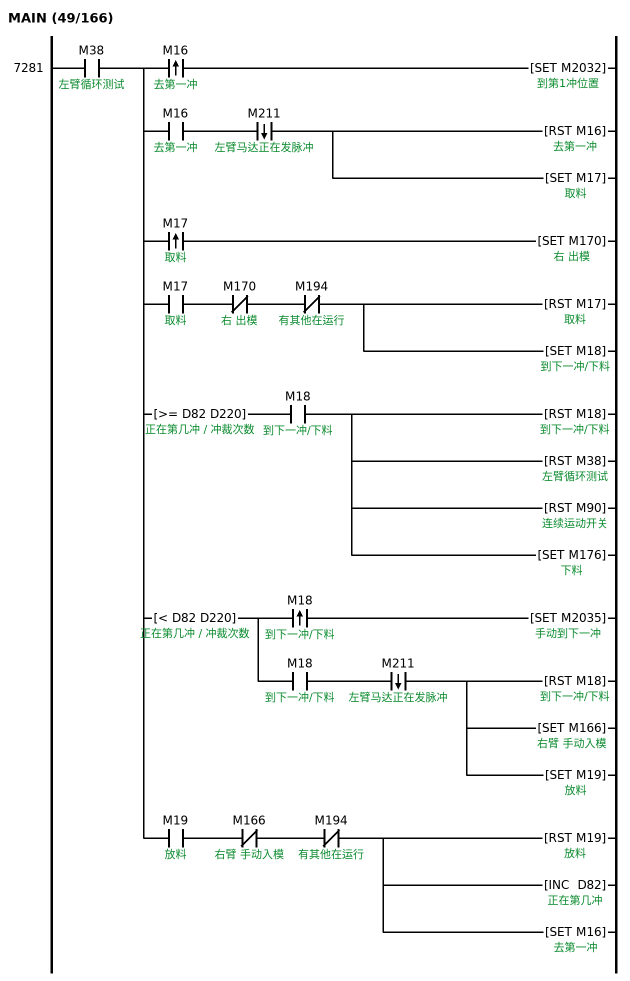
[picture p48: ladder of MAIN, rungs at steps 7281 to 7281]
7281  LD      M38  ; 左臂循环测试
      MPS
      ANDP    M16  ; 去第一冲
      SET     M2032  ; 到第1冲位置
      MRD
      AND     M16  ; 去第一冲
      ANDF    M211  ; 左臂马达正在发脉冲
      RST     M16  ; 去第一冲
      SET     M17  ; 取料
      MRD
      ANDP    M17  ; 取料
      SET     M170  ; 右 出模
      MRD
      AND     M17  ; 取料
      ANI     M170  ; 右 出模
      ANI     M194  ; 有其他在运行
      RST     M17  ; 取料
      SET     M18  ; 到下一冲/下料
      MRD
      AND>=   D82 D220  ; 正在第几冲 / 冲裁次数
      AND     M18  ; 到下一冲/下料
      RST     M18  ; 到下一冲/下料
      RST     M38  ; 左臂循环测试
      RST     M90  ; 连续运动开关
      SET     M176  ; 下料
      MRD
      AND<    D82 D220  ; 正在第几冲 / 冲裁次数
      MPS
      ANDP    M18  ; 到下一冲/下料
      SET     M2035  ; 手动到下一冲
      MPP
      AND     M18  ; 到下一冲/下料
      ANDF    M211  ; 左臂马达正在发脉冲
      RST     M18  ; 到下一冲/下料
      SET     M166  ; 右臂 手动入模
      SET     M19  ; 放料
      MPP
      AND     M19  ; 放料
      ANI     M166  ; 右臂 手动入模
      ANI     M194  ; 有其他在运行
      RST     M19  ; 放料
      INC     D82
      SET     M16  ; 去第一冲
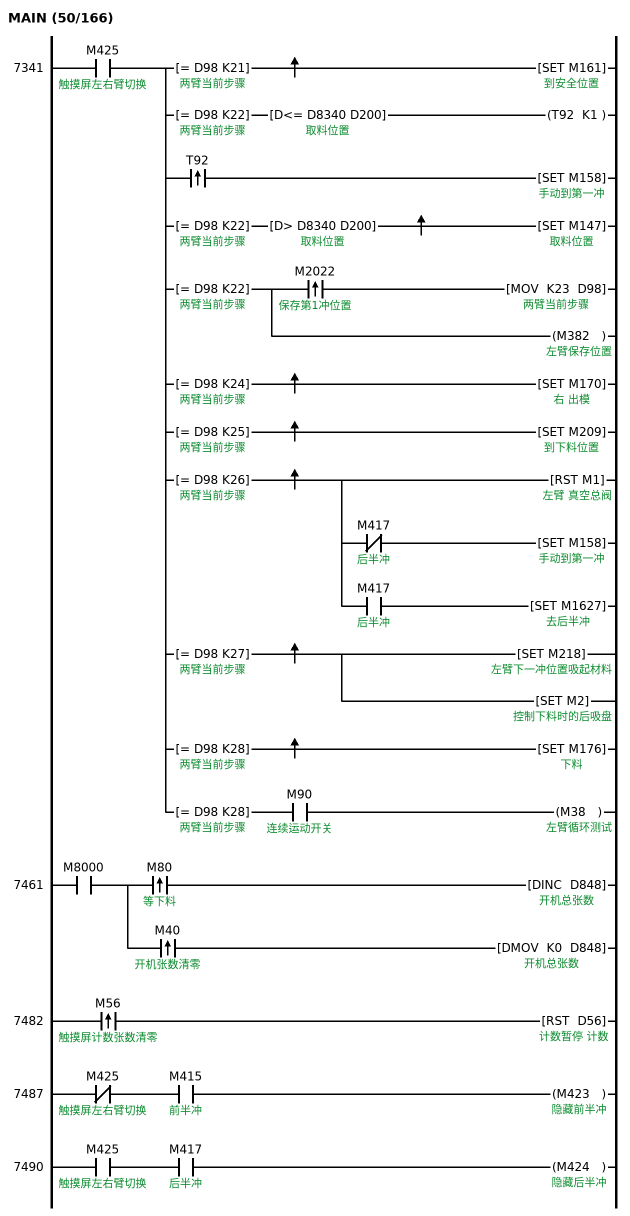
7341  LD      M425  ; 触摸屏左右臂切换
      MPS
      AND=    D98 K21  ; 两臂当前步骤
      MEP
      SET     M161  ; 到安全位置
      MRD
      AND=    D98 K22  ; 两臂当前步骤
      ANDD<=  D8340 D200  ; 取料位置
      OUT     T92 K1
      MRD
      ANDP    T92
      SET     M158  ; 手动到第一冲
      MRD
      AND=    D98 K22  ; 两臂当前步骤
      ANDD>   D8340 D200  ; 取料位置
      MEP
      SET     M147  ; 取料位置
      MRD
      AND=    D98 K22  ; 两臂当前步骤
      MPS
      ANDP    M2022  ; 保存第1冲位置
      MOV     K23 D98
      MPP
      OUT     M382  ; 左臂保存位置
      MRD
      AND=    D98 K24  ; 两臂当前步骤
      MEP
      SET     M170  ; 右 出模
      MRD
      AND=    D98 K25  ; 两臂当前步骤
      MEP
      SET     M209  ; 到下料位置
      MRD
      AND=    D98 K26  ; 两臂当前步骤
      MEP
      RST     M1  ; 左臂 真空总阀
      MPS
      ANI     M417  ; 后半冲
      SET     M158  ; 手动到第一冲
      MPP
      AND     M417  ; 后半冲
      SET     M1627  ; 去后半冲
      MRD
      AND=    D98 K27  ; 两臂当前步骤
      MEP
      SET     M218  ; 左臂下一冲位置吸起材料
      SET     M2  ; 控制下料时的后吸盘
      MRD
      AND=    D98 K28  ; 两臂当前步骤
      MEP
      SET     M176  ; 下料
      MPP
      AND=    D98 K28  ; 两臂当前步骤
      AND     M90  ; 连续运动开关
      OUT     M38  ; 左臂循环测试
7461  LD      M8000
      MPS
      ANDP    M80  ; 等下料
      DINC    D848
      MPP
      ANDP    M40  ; 开机张数清零
      DMOV    K0 D848
7482  LDP     M56  ; 触摸屏计数张数清零
      RST     D56  ; 计数暂停 计数
7487  LDI     M425  ; 触摸屏左右臂切换
      AND     M415  ; 前半冲
      OUT     M423  ; 隐藏前半冲
7490  LD      M425  ; 触摸屏左右臂切换
      AND     M417  ; 后半冲
      OUT     M424  ; 隐藏后半冲
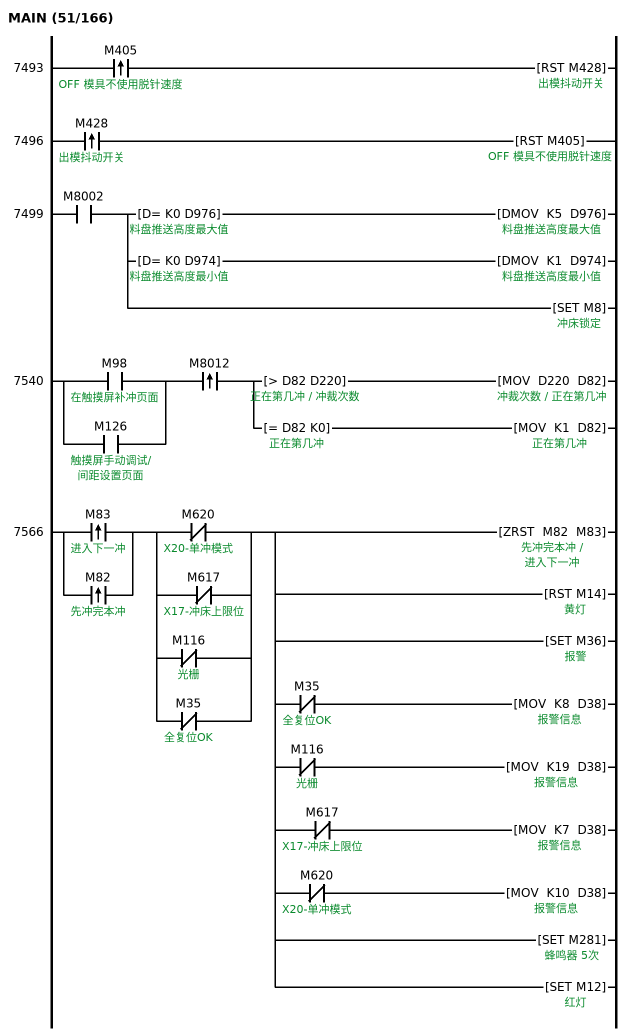
7493  LDP     M405  ; OFF 模具不使用脱针速度
      RST     M428  ; 出模抖动开关
7496  LDP     M428  ; 出模抖动开关
      RST     M405  ; OFF 模具不使用脱针速度
7499  LD      M8002
      MPS
      ANDD=   K0 D976  ; 料盘推送高度最大值
      DMOV    K5 D976
      MRD
      ANDD=   K0 D974  ; 料盘推送高度最小值
      DMOV    K1 D974
      MPP
      SET     M8  ; 冲床锁定
7540  LD      M98  ; 在触摸屏补冲页面
      OR      M126  ; 触摸屏手动调试/间距设置页面
      ANDP    M8012
      MPS
      AND>    D82 D220  ; 正在第几冲 / 冲裁次数
      MOV     D220 D82
      MPP
      AND=    D82 K0  ; 正在第几冲
      MOV     K1 D82
7566  LDP     M83  ; 进入下一冲
      ORP     M82  ; 先冲完本冲
      LDI     M620  ; X20-单冲模式
      ORI     M617  ; X17-冲床上限位
      ORI     M116  ; 光栅
      ORI     M35  ; 全复位OK
      ANB
      ZRST    M82 M83
      RST     M14  ; 黄灯
      SET     M36  ; 报警
      MPS
      ANI     M35  ; 全复位OK
      MOV     K8 D38
      MRD
      ANI     M116  ; 光栅
      MOV     K19 D38
      MRD
      ANI     M617  ; X17-冲床上限位
      MOV     K7 D38
      MRD
      ANI     M620  ; X20-单冲模式
      MOV     K10 D38
      MPP
      SET     M281  ; 蜂鸣器 5次
      SET     M12  ; 红灯
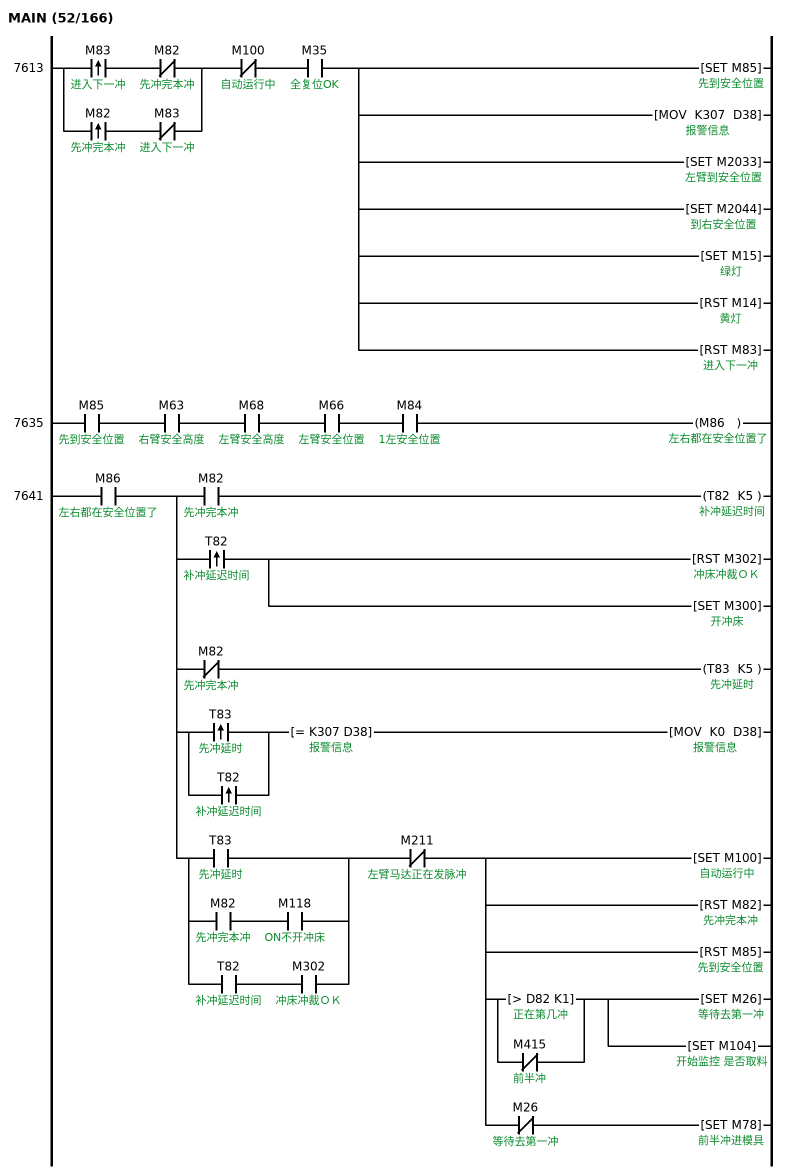
7613  LDP     M83  ; 进入下一冲
      ANI     M82  ; 先冲完本冲
      LDP     M82  ; 先冲完本冲
      ANI     M83  ; 进入下一冲
      ORB
      ANI     M100  ; 自动运行中
      AND     M35  ; 全复位OK
      SET     M85  ; 先到安全位置
      MOV     K307 D38
      SET     M2033  ; 左臂到安全位置
      SET     M2044  ; 到右安全位置
      SET     M15  ; 绿灯
      RST     M14  ; 黄灯
      RST     M83  ; 进入下一冲
7635  LD      M85  ; 先到安全位置
      AND     M63  ; 右臂安全高度
      AND     M68  ; 左臂安全高度
      AND     M66  ; 左臂安全位置
      AND     M84  ; 1左安全位置
      OUT     M86  ; 左右都在安全位置了
7641  LD      M86  ; 左右都在安全位置了
      MPS
      AND     M82  ; 先冲完本冲
      OUT     T82 K5  ; 补冲延迟时间
      MRD
      ANDP    T82  ; 补冲延迟时间
      RST     M302  ; 冲床冲裁ＯＫ
      SET     M300  ; 开冲床
      MRD
      ANI     M82  ; 先冲完本冲
      OUT     T83 K5  ; 先冲延时
      MRD
      LDP     T83  ; 先冲延时
      ORP     T82  ; 补冲延迟时间
      ANB
      AND=    K307 D38  ; 报警信息
      MOV     K0 D38
      MPP
      LD      T83  ; 先冲延时
      LD      M82  ; 先冲完本冲
      AND     M118  ; ON不开冲床
      ORB
      LD      T82  ; 补冲延迟时间
      AND     M302  ; 冲床冲裁ＯＫ
      ORB
      ANB
      ANI     M211  ; 左臂马达正在发脉冲
      SET     M100  ; 自动运行中
      RST     M82  ; 先冲完本冲
      RST     M85  ; 先到安全位置
      MPS
      LD>     D82 K1  ; 正在第几冲
      ORI     M415  ; 前半冲
      ANB
      SET     M26  ; 等待去第一冲
      SET     M104  ; 开始监控 是否取料
      MPP
      ANI     M26  ; 等待去第一冲
      SET     M78  ; 前半冲进模具
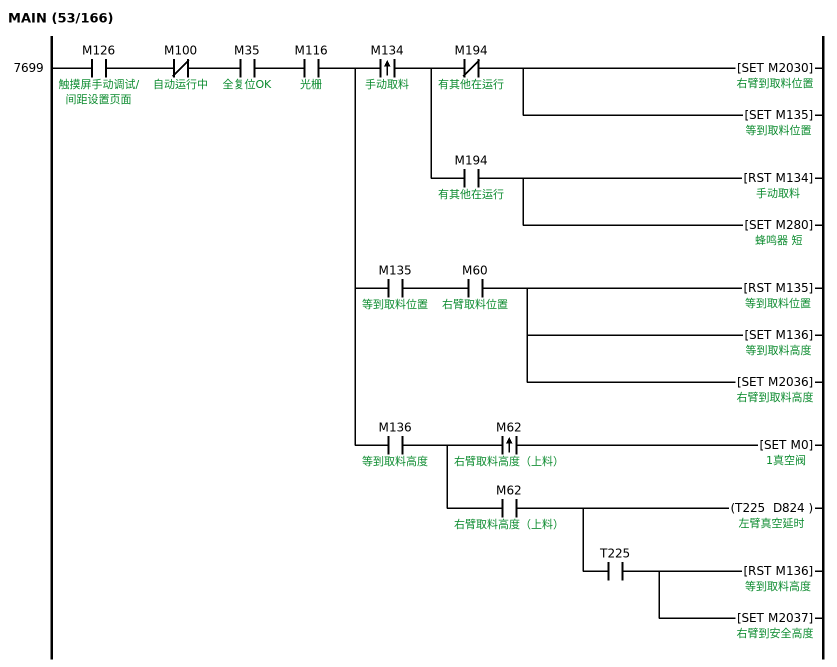
7699  LD      M126  ; 触摸屏手动调试/间距设置页面
      ANI     M100  ; 自动运行中
      AND     M35  ; 全复位OK
      AND     M116  ; 光栅
      MPS
      ANDP    M134  ; 手动取料
      MPS
      ANI     M194  ; 有其他在运行
      SET     M2030  ; 右臂到取料位置
      SET     M135  ; 等到取料位置
      MPP
      AND     M194  ; 有其他在运行
      RST     M134  ; 手动取料
      SET     M280  ; 蜂鸣器 短
      MRD
      AND     M135  ; 等到取料位置
      AND     M60  ; 右臂取料位置
      RST     M135  ; 等到取料位置
      SET     M136  ; 等到取料高度
      SET     M2036  ; 右臂到取料高度
      MPP
      AND     M136  ; 等到取料高度
      MPS
      ANDP    M62  ; 右臂取料高度（上料）
      SET     M0  ; 1真空阀
      MPP
      AND     M62  ; 右臂取料高度（上料）
      OUT     T225 D824  ; 左臂真空延时
      AND     T225
      RST     M136  ; 等到取料高度
      SET     M2037  ; 右臂到安全高度
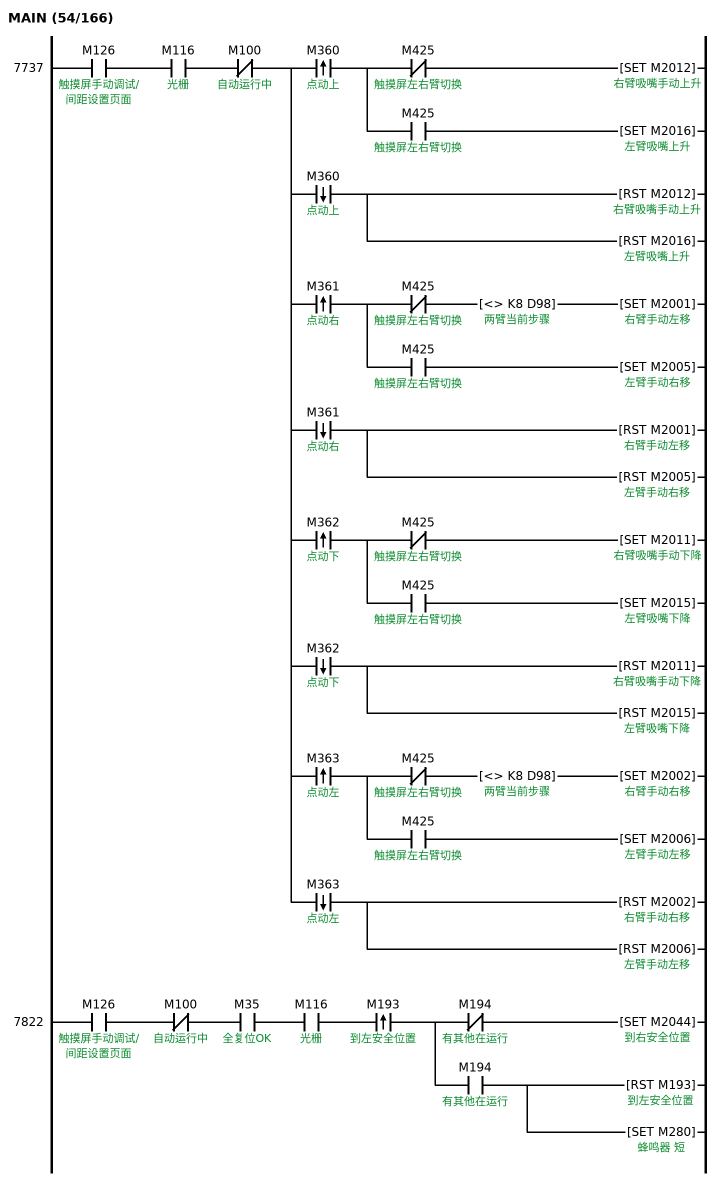
7737  LD      M126  ; 触摸屏手动调试/间距设置页面
      AND     M116  ; 光栅
      ANI     M100  ; 自动运行中
      MPS
      ANDP    M360  ; 点动上
      MPS
      ANI     M425  ; 触摸屏左右臂切换
      SET     M2012  ; 右臂吸嘴手动上升
      MPP
      AND     M425  ; 触摸屏左右臂切换
      SET     M2016  ; 左臂吸嘴上升
      MRD
      ANDF    M360  ; 点动上
      RST     M2012  ; 右臂吸嘴手动上升
      RST     M2016  ; 左臂吸嘴上升
      MRD
      ANDP    M361  ; 点动右
      MPS
      ANI     M425  ; 触摸屏左右臂切换
      AND<>   K8 D98  ; 两臂当前步骤
      SET     M2001  ; 右臂手动左移
      MPP
      AND     M425  ; 触摸屏左右臂切换
      SET     M2005  ; 左臂手动右移
      MRD
      ANDF    M361  ; 点动右
      RST     M2001  ; 右臂手动左移
      RST     M2005  ; 左臂手动右移
      MRD
      ANDP    M362  ; 点动下
      MPS
      ANI     M425  ; 触摸屏左右臂切换
      SET     M2011  ; 右臂吸嘴手动下降
      MPP
      AND     M425  ; 触摸屏左右臂切换
      SET     M2015  ; 左臂吸嘴下降
      MRD
      ANDF    M362  ; 点动下
      RST     M2011  ; 右臂吸嘴手动下降
      RST     M2015  ; 左臂吸嘴下降
      MRD
      ANDP    M363  ; 点动左
      MPS
      ANI     M425  ; 触摸屏左右臂切换
      AND<>   K8 D98  ; 两臂当前步骤
      SET     M2002  ; 右臂手动右移
      MPP
      AND     M425  ; 触摸屏左右臂切换
      SET     M2006  ; 左臂手动左移
      MPP
      ANDF    M363  ; 点动左
      RST     M2002  ; 右臂手动右移
      RST     M2006  ; 左臂手动左移
7822  LD      M126  ; 触摸屏手动调试/间距设置页面
      ANI     M100  ; 自动运行中
      AND     M35  ; 全复位OK
      AND     M116  ; 光栅
      ANDP    M193  ; 到左安全位置
      MPS
      ANI     M194  ; 有其他在运行
      SET     M2044  ; 到右安全位置
      MPP
      AND     M194  ; 有其他在运行
      RST     M193  ; 到左安全位置
      SET     M280  ; 蜂鸣器 短
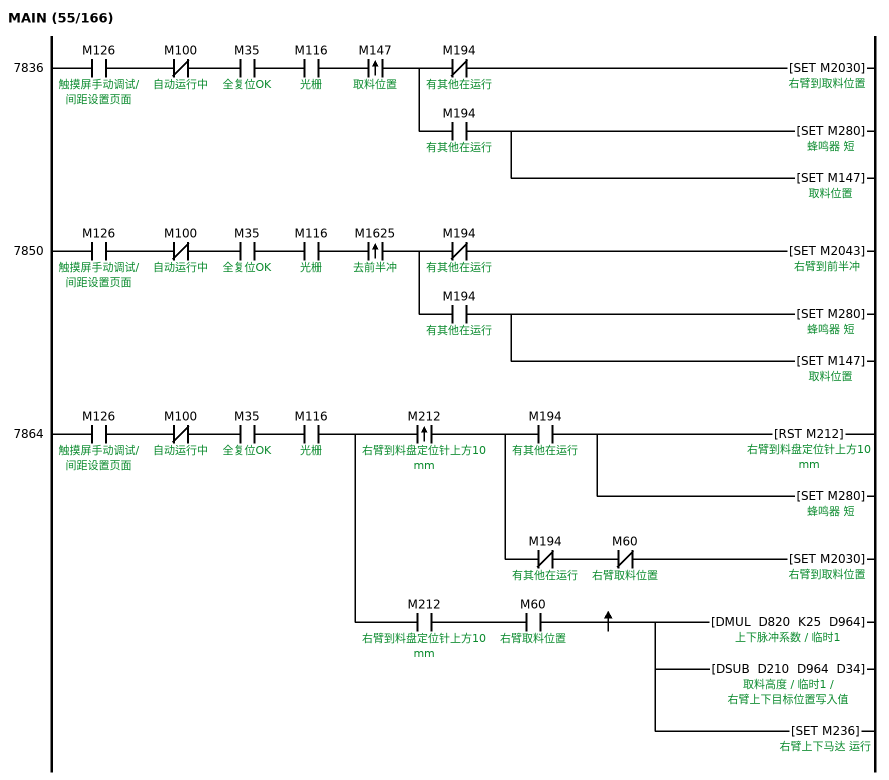
7836  LD      M126  ; 触摸屏手动调试/间距设置页面
      ANI     M100  ; 自动运行中
      AND     M35  ; 全复位OK
      AND     M116  ; 光栅
      ANDP    M147  ; 取料位置
      MPS
      ANI     M194  ; 有其他在运行
      SET     M2030  ; 右臂到取料位置
      MPP
      AND     M194  ; 有其他在运行
      SET     M280  ; 蜂鸣器 短
      SET     M147  ; 取料位置
7850  LD      M126  ; 触摸屏手动调试/间距设置页面
      ANI     M100  ; 自动运行中
      AND     M35  ; 全复位OK
      AND     M116  ; 光栅
      ANDP    M1625  ; 去前半冲
      MPS
      ANI     M194  ; 有其他在运行
      SET     M2043  ; 右臂到前半冲
      MPP
      AND     M194  ; 有其他在运行
      SET     M280  ; 蜂鸣器 短
      SET     M147  ; 取料位置
7864  LD      M126  ; 触摸屏手动调试/间距设置页面
      ANI     M100  ; 自动运行中
      AND     M35  ; 全复位OK
      AND     M116  ; 光栅
      MPS
      ANDP    M212  ; 右臂到料盘定位针上方10mm
      MPS
      AND     M194  ; 有其他在运行
      RST     M212  ; 右臂到料盘定位针上方10mm
      SET     M280  ; 蜂鸣器 短
      MPP
      ANI     M194  ; 有其他在运行
      ANI     M60  ; 右臂取料位置
      SET     M2030  ; 右臂到取料位置
      MPP
      AND     M212  ; 右臂到料盘定位针上方10mm
      AND     M60  ; 右臂取料位置
      MEP
      DMUL    D820 K25 D964
      DSUB    D210 D964 D34  ; 右臂上下目标位置写入值
      SET     M236  ; 右臂上下马达 运行
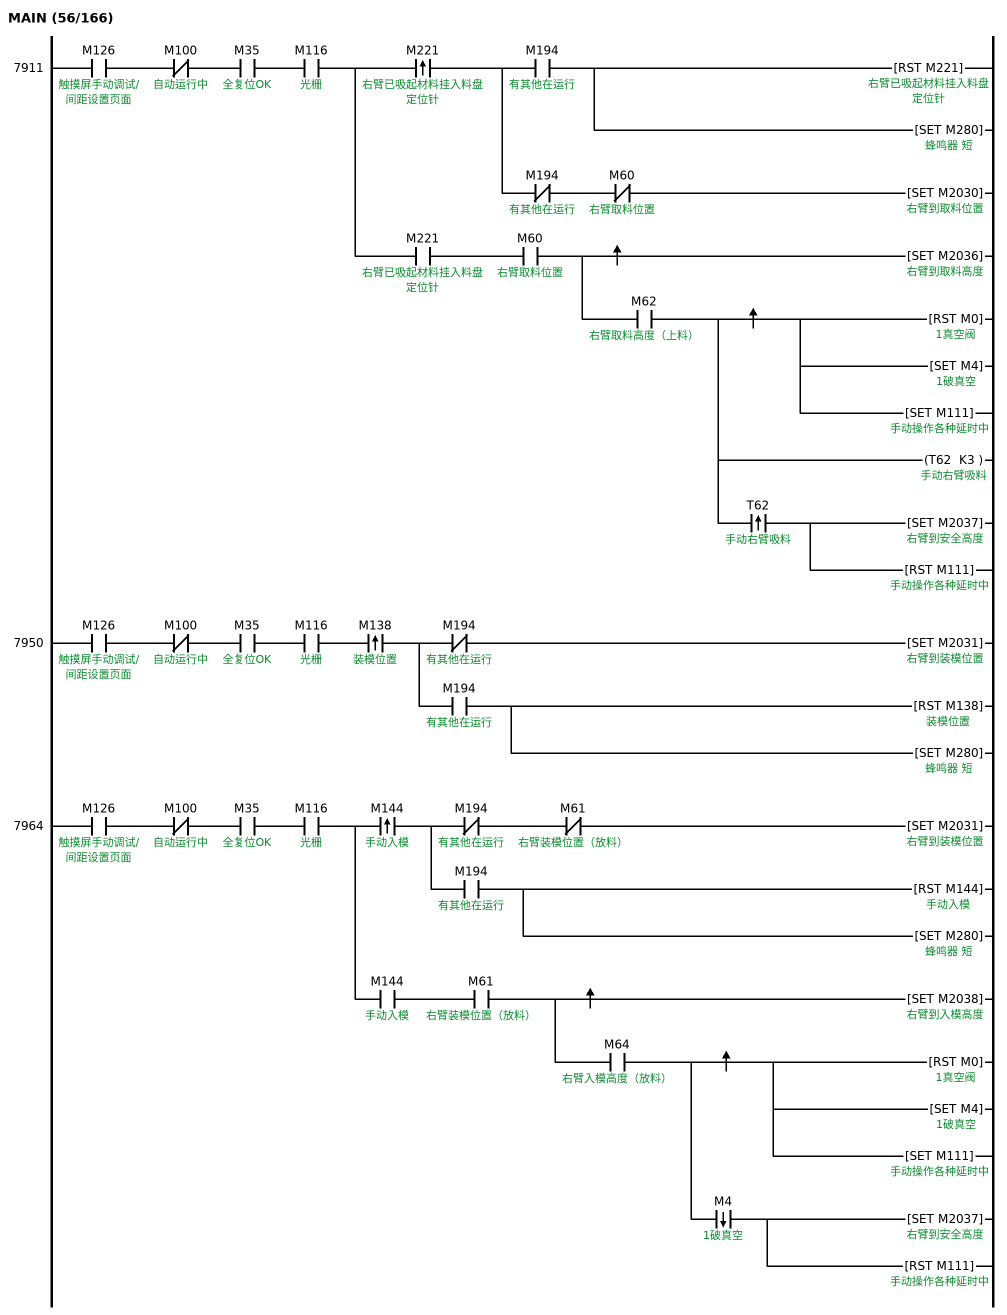
7911  LD      M126  ; 触摸屏手动调试/间距设置页面
      ANI     M100  ; 自动运行中
      AND     M35  ; 全复位OK
      AND     M116  ; 光栅
      MPS
      ANDP    M221  ; 右臂已吸起材料挂入料盘定位针
      MPS
      AND     M194  ; 有其他在运行
      RST     M221  ; 右臂已吸起材料挂入料盘定位针
      SET     M280  ; 蜂鸣器 短
      MPP
      ANI     M194  ; 有其他在运行
      ANI     M60  ; 右臂取料位置
      SET     M2030  ; 右臂到取料位置
      MPP
      AND     M221  ; 右臂已吸起材料挂入料盘定位针
      AND     M60  ; 右臂取料位置
      MPS
      MEP
      SET     M2036  ; 右臂到取料高度
      MPP
      AND     M62  ; 右臂取料高度（上料）
      MPS
      MEP
      RST     M0  ; 1真空阀
      SET     M4  ; 1破真空
      SET     M111  ; 手动操作各种延时中
      MPP
      OUT     T62 K3  ; 手动右臂吸料
      ANDP    T62  ; 手动右臂吸料
      SET     M2037  ; 右臂到安全高度
      RST     M111  ; 手动操作各种延时中
7950  LD      M126  ; 触摸屏手动调试/间距设置页面
      ANI     M100  ; 自动运行中
      AND     M35  ; 全复位OK
      AND     M116  ; 光栅
      ANDP    M138  ; 装模位置
      MPS
      ANI     M194  ; 有其他在运行
      SET     M2031  ; 右臂到装模位置
      MPP
      AND     M194  ; 有其他在运行
      RST     M138  ; 装模位置
      SET     M280  ; 蜂鸣器 短
7964  LD      M126  ; 触摸屏手动调试/间距设置页面
      ANI     M100  ; 自动运行中
      AND     M35  ; 全复位OK
      AND     M116  ; 光栅
      MPS
      ANDP    M144  ; 手动入模
      MPS
      ANI     M194  ; 有其他在运行
      ANI     M61  ; 右臂装模位置（放料）
      SET     M2031  ; 右臂到装模位置
      MPP
      AND     M194  ; 有其他在运行
      RST     M144  ; 手动入模
      SET     M280  ; 蜂鸣器 短
      MPP
      AND     M144  ; 手动入模
      AND     M61  ; 右臂装模位置（放料）
      MPS
      MEP
      SET     M2038  ; 右臂到入模高度
      MPP
      AND     M64  ; 右臂入模高度（放料）
      MPS
      MEP
      RST     M0  ; 1真空阀
      SET     M4  ; 1破真空
      SET     M111  ; 手动操作各种延时中
      MPP
      ANDF    M4  ; 1破真空
      SET     M2037  ; 右臂到安全高度
      RST     M111  ; 手动操作各种延时中
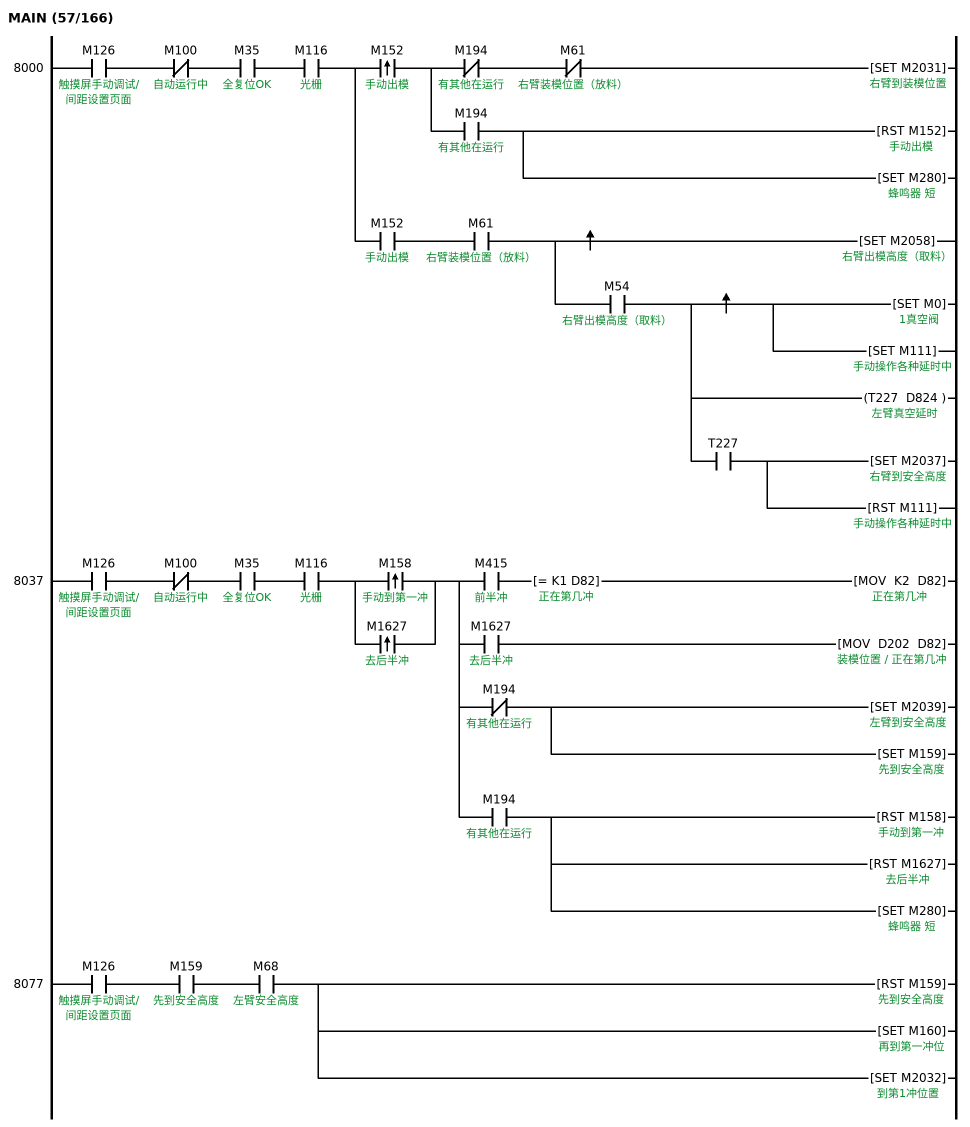
8000  LD      M126  ; 触摸屏手动调试/间距设置页面
      ANI     M100  ; 自动运行中
      AND     M35  ; 全复位OK
      AND     M116  ; 光栅
      MPS
      ANDP    M152  ; 手动出模
      MPS
      ANI     M194  ; 有其他在运行
      ANI     M61  ; 右臂装模位置（放料）
      SET     M2031  ; 右臂到装模位置
      MPP
      AND     M194  ; 有其他在运行
      RST     M152  ; 手动出模
      SET     M280  ; 蜂鸣器 短
      MPP
      AND     M152  ; 手动出模
      AND     M61  ; 右臂装模位置（放料）
      MPS
      MEP
      SET     M2058  ; 右臂出模高度（取料）
      MPP
      AND     M54  ; 右臂出模高度（取料）
      MPS
      MEP
      SET     M0  ; 1真空阀
      SET     M111  ; 手动操作各种延时中
      MPP
      OUT     T227 D824  ; 左臂真空延时
      AND     T227
      SET     M2037  ; 右臂到安全高度
      RST     M111  ; 手动操作各种延时中
8037  LD      M126  ; 触摸屏手动调试/间距设置页面
      ANI     M100  ; 自动运行中
      AND     M35  ; 全复位OK
      AND     M116  ; 光栅
      LDP     M158  ; 手动到第一冲
      ORP     M1627  ; 去后半冲
      ANB
      MPS
      AND     M415  ; 前半冲
      AND=    K1 D82  ; 正在第几冲
      MOV     K2 D82
      MRD
      AND     M1627  ; 去后半冲
      MOV     D202 D82
      MRD
      ANI     M194  ; 有其他在运行
      SET     M2039  ; 左臂到安全高度
      SET     M159  ; 先到安全高度
      MPP
      AND     M194  ; 有其他在运行
      RST     M158  ; 手动到第一冲
      RST     M1627  ; 去后半冲
      SET     M280  ; 蜂鸣器 短
8077  LD      M126  ; 触摸屏手动调试/间距设置页面
      AND     M159  ; 先到安全高度
      AND     M68  ; 左臂安全高度
      RST     M159  ; 先到安全高度
      SET     M160  ; 再到第一冲位
      SET     M2032  ; 到第1冲位置
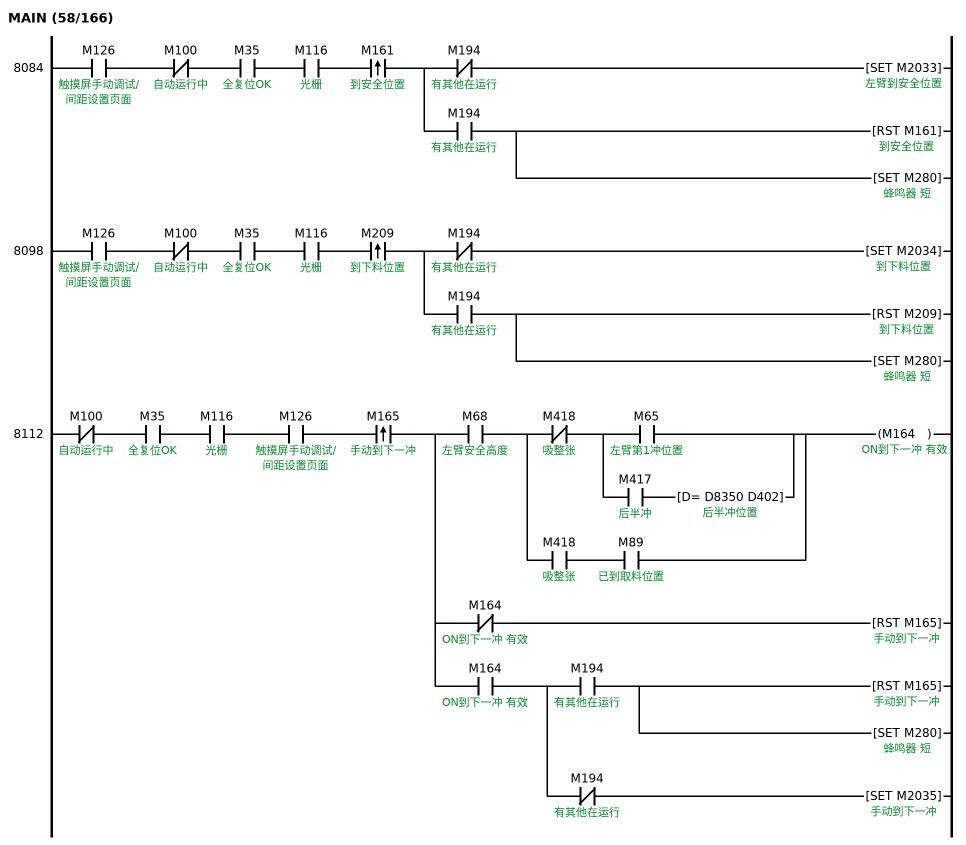
8084  LD      M126  ; 触摸屏手动调试/间距设置页面
      ANI     M100  ; 自动运行中
      AND     M35  ; 全复位OK
      AND     M116  ; 光栅
      ANDP    M161  ; 到安全位置
      MPS
      ANI     M194  ; 有其他在运行
      SET     M2033  ; 左臂到安全位置
      MPP
      AND     M194  ; 有其他在运行
      RST     M161  ; 到安全位置
      SET     M280  ; 蜂鸣器 短
8098  LD      M126  ; 触摸屏手动调试/间距设置页面
      ANI     M100  ; 自动运行中
      AND     M35  ; 全复位OK
      AND     M116  ; 光栅
      ANDP    M209  ; 到下料位置
      MPS
      ANI     M194  ; 有其他在运行
      SET     M2034  ; 到下料位置
      MPP
      AND     M194  ; 有其他在运行
      RST     M209  ; 到下料位置
      SET     M280  ; 蜂鸣器 短
8112  LDI     M100  ; 自动运行中
      AND     M35  ; 全复位OK
      AND     M116  ; 光栅
      AND     M126  ; 触摸屏手动调试/间距设置页面
      ANDP    M165  ; 手动到下一冲
      MPS
      AND     M68  ; 左臂安全高度
      LDI     M418  ; 吸整张
      LD      M65  ; 左臂第1冲位置
      LD      M417  ; 后半冲
      ANDD=   D8350 D402  ; 后半冲位置
      ORB
      ANB
      LD      M418  ; 吸整张
      AND     M89  ; 已到取料位置
      ORB
      ANB
      OUT     M164  ; ON到下一冲 有效
      MRD
      ANI     M164  ; ON到下一冲 有效
      RST     M165  ; 手动到下一冲
      MPP
      AND     M164  ; ON到下一冲 有效
      MPS
      AND     M194  ; 有其他在运行
      RST     M165  ; 手动到下一冲
      SET     M280  ; 蜂鸣器 短
      MPP
      ANI     M194  ; 有其他在运行
      SET     M2035  ; 手动到下一冲
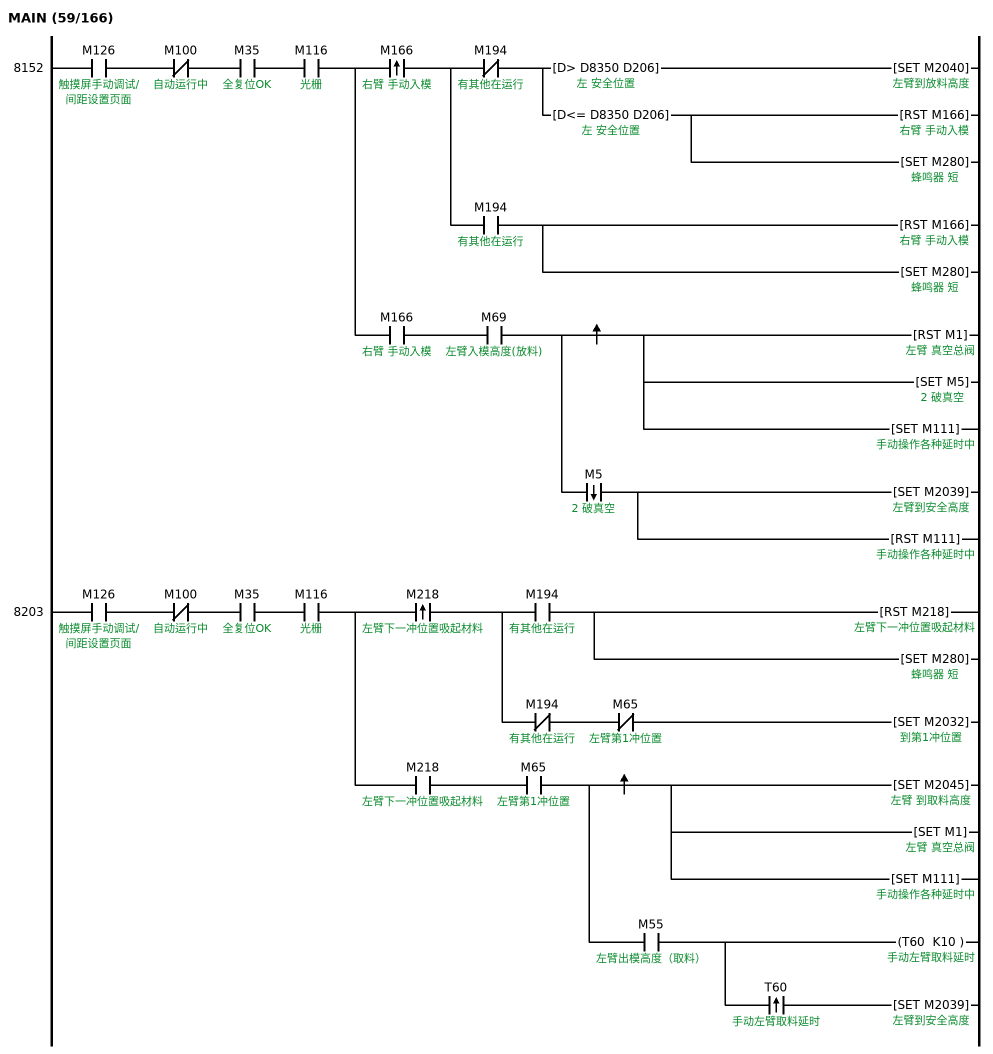
8152  LD      M126  ; 触摸屏手动调试/间距设置页面
      ANI     M100  ; 自动运行中
      AND     M35  ; 全复位OK
      AND     M116  ; 光栅
      MPS
      ANDP    M166  ; 右臂 手动入模
      MPS
      ANI     M194  ; 有其他在运行
      MPS
      ANDD>   D8350 D206  ; 左 安全位置
      SET     M2040  ; 左臂到放料高度
      MPP
      ANDD<=  D8350 D206  ; 左 安全位置
      RST     M166  ; 右臂 手动入模
      SET     M280  ; 蜂鸣器 短
      MPP
      AND     M194  ; 有其他在运行
      RST     M166  ; 右臂 手动入模
      SET     M280  ; 蜂鸣器 短
      MPP
      AND     M166  ; 右臂 手动入模
      AND     M69  ; 左臂入模高度(放料)
      MPS
      MEP
      RST     M1  ; 左臂 真空总阀
      SET     M5  ; 2 破真空
      SET     M111  ; 手动操作各种延时中
      MPP
      ANDF    M5  ; 2 破真空
      SET     M2039  ; 左臂到安全高度
      RST     M111  ; 手动操作各种延时中
8203  LD      M126  ; 触摸屏手动调试/间距设置页面
      ANI     M100  ; 自动运行中
      AND     M35  ; 全复位OK
      AND     M116  ; 光栅
      MPS
      ANDP    M218  ; 左臂下一冲位置吸起材料
      MPS
      AND     M194  ; 有其他在运行
      RST     M218  ; 左臂下一冲位置吸起材料
      SET     M280  ; 蜂鸣器 短
      MPP
      ANI     M194  ; 有其他在运行
      ANI     M65  ; 左臂第1冲位置
      SET     M2032  ; 到第1冲位置
      MPP
      AND     M218  ; 左臂下一冲位置吸起材料
      AND     M65  ; 左臂第1冲位置
      MPS
      MEP
      SET     M2045  ; 左臂 到取料高度
      SET     M1  ; 左臂 真空总阀
      SET     M111  ; 手动操作各种延时中
      MPP
      AND     M55  ; 左臂出模高度（取料）
      OUT     T60 K10  ; 手动左臂取料延时
      ANDP    T60  ; 手动左臂取料延时
      SET     M2039  ; 左臂到安全高度
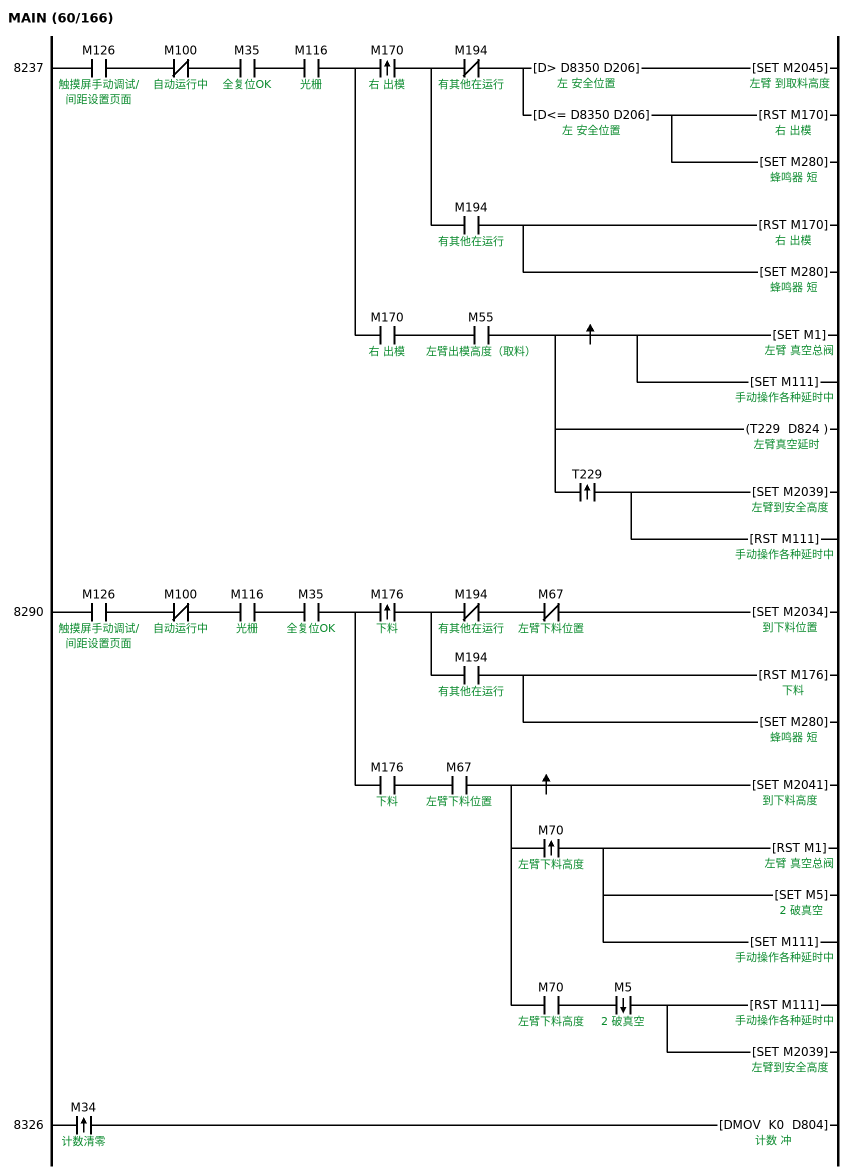
8237  LD      M126  ; 触摸屏手动调试/间距设置页面
      ANI     M100  ; 自动运行中
      AND     M35  ; 全复位OK
      AND     M116  ; 光栅
      MPS
      ANDP    M170  ; 右 出模
      MPS
      ANI     M194  ; 有其他在运行
      MPS
      ANDD>   D8350 D206  ; 左 安全位置
      SET     M2045  ; 左臂 到取料高度
      MPP
      ANDD<=  D8350 D206  ; 左 安全位置
      RST     M170  ; 右 出模
      SET     M280  ; 蜂鸣器 短
      MPP
      AND     M194  ; 有其他在运行
      RST     M170  ; 右 出模
      SET     M280  ; 蜂鸣器 短
      MPP
      AND     M170  ; 右 出模
      AND     M55  ; 左臂出模高度（取料）
      MPS
      MEP
      SET     M1  ; 左臂 真空总阀
      SET     M111  ; 手动操作各种延时中
      MPP
      OUT     T229 D824  ; 左臂真空延时
      ANDP    T229
      SET     M2039  ; 左臂到安全高度
      RST     M111  ; 手动操作各种延时中
8290  LD      M126  ; 触摸屏手动调试/间距设置页面
      ANI     M100  ; 自动运行中
      AND     M116  ; 光栅
      AND     M35  ; 全复位OK
      MPS
      ANDP    M176  ; 下料
      MPS
      ANI     M194  ; 有其他在运行
      ANI     M67  ; 左臂下料位置
      SET     M2034  ; 到下料位置
      MPP
      AND     M194  ; 有其他在运行
      RST     M176  ; 下料
      SET     M280  ; 蜂鸣器 短
      MPP
      AND     M176  ; 下料
      AND     M67  ; 左臂下料位置
      MPS
      MEP
      SET     M2041  ; 到下料高度
      MRD
      ANDP    M70  ; 左臂下料高度
      RST     M1  ; 左臂 真空总阀
      SET     M5  ; 2 破真空
      SET     M111  ; 手动操作各种延时中
      MPP
      AND     M70  ; 左臂下料高度
      ANDF    M5  ; 2 破真空
      RST     M111  ; 手动操作各种延时中
      SET     M2039  ; 左臂到安全高度
8326  LDP     M34  ; 计数清零
      DMOV    K0 D804
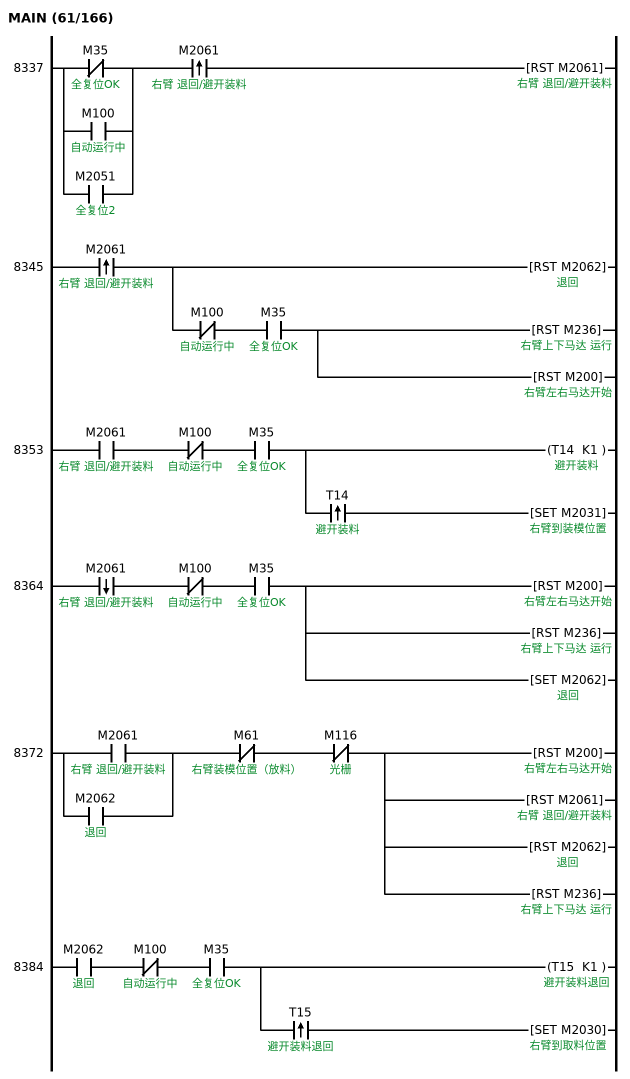
8337  LDI     M35  ; 全复位OK
      OR      M100  ; 自动运行中
      OR      M2051  ; 全复位2
      ANDP    M2061  ; 右臂 退回/避开装料
      RST     M2061  ; 右臂 退回/避开装料
8345  LDP     M2061  ; 右臂 退回/避开装料
      RST     M2062  ; 退回
      ANI     M100  ; 自动运行中
      AND     M35  ; 全复位OK
      RST     M236  ; 右臂上下马达 运行
      RST     M200  ; 右臂左右马达开始
8353  LD      M2061  ; 右臂 退回/避开装料
      ANI     M100  ; 自动运行中
      AND     M35  ; 全复位OK
      OUT     T14 K1  ; 避开装料
      ANDP    T14  ; 避开装料
      SET     M2031  ; 右臂到装模位置
8364  LDF     M2061  ; 右臂 退回/避开装料
      ANI     M100  ; 自动运行中
      AND     M35  ; 全复位OK
      RST     M200  ; 右臂左右马达开始
      RST     M236  ; 右臂上下马达 运行
      SET     M2062  ; 退回
8372  LD      M2061  ; 右臂 退回/避开装料
      OR      M2062  ; 退回
      ANI     M61  ; 右臂装模位置（放料）
      ANI     M116  ; 光栅
      RST     M200  ; 右臂左右马达开始
      RST     M2061  ; 右臂 退回/避开装料
      RST     M2062  ; 退回
      RST     M236  ; 右臂上下马达 运行
8384  LD      M2062  ; 退回
      ANI     M100  ; 自动运行中
      AND     M35  ; 全复位OK
      OUT     T15 K1  ; 避开装料退回
      ANDP    T15  ; 避开装料退回
      SET     M2030  ; 右臂到取料位置
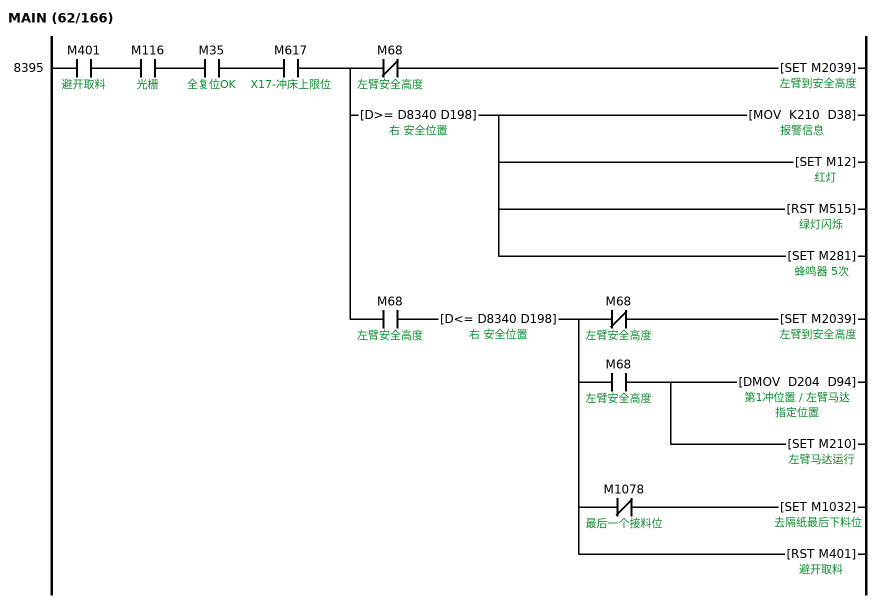
8395  LD      M401  ; 避开取料
      AND     M116  ; 光栅
      AND     M35  ; 全复位OK
      AND     M617  ; X17-冲床上限位
      MPS
      ANI     M68  ; 左臂安全高度
      SET     M2039  ; 左臂到安全高度
      MRD
      ANDD>=  D8340 D198  ; 右 安全位置
      MOV     K210 D38
      SET     M12  ; 红灯
      RST     M515  ; 绿灯闪烁
      SET     M281  ; 蜂鸣器 5次
      MPP
      AND     M68  ; 左臂安全高度
      ANDD<=  D8340 D198  ; 右 安全位置
      MPS
      ANI     M68  ; 左臂安全高度
      SET     M2039  ; 左臂到安全高度
      MRD
      AND     M68  ; 左臂安全高度
      DMOV    D204 D94
      SET     M210  ; 左臂马达运行
      MRD
      ANI     M1078  ; 最后一个接料位
      SET     M1032  ; 去隔纸最后下料位
      MPP
      RST     M401  ; 避开取料
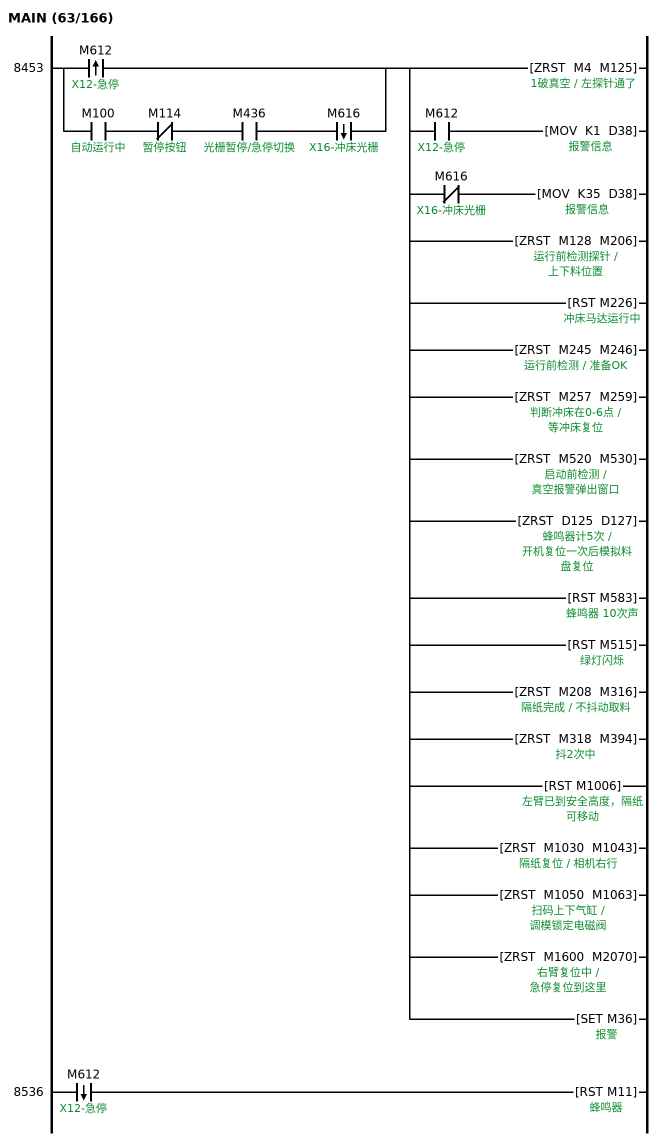
8453  LDP     M612  ; X12-急停
      LD      M100  ; 自动运行中
      ANI     M114  ; 暂停按钮
      AND     M436  ; 光栅暂停/急停切换
      ANDF    M616  ; X16-冲床光栅
      ORB
      ZRST    M4 M125
      MPS
      AND     M612  ; X12-急停
      MOV     K1 D38
      MRD
      ANI     M616  ; X16-冲床光栅
      MOV     K35 D38
      MPP
      ZRST    M128 M206  ; 上下料位置
      RST     M226  ; 冲床马达运行中
      ZRST    M245 M246  ; 运行前检测 / 准备OK
      ZRST    M257 M259  ; 判断冲床在0-6点 / 等冲床复位
      ZRST    M520 M530  ; 启动前检测
      ZRST    D125 D127  ; 蜂鸣器计5次 / 开机复位一次后模拟料盘复位
      RST     M583  ; 蜂鸣器 10次声
      RST     M515  ; 绿灯闪烁
      ZRST    M208 M316  ; 隔纸完成
      ZRST    M318 M394
      RST     M1006  ; 左臂已到安全高度，隔纸可移动
      ZRST    M1030 M1043
      ZRST    M1050 M1063
      ZRST    M1600 M2070  ; 急停复位到这里
      SET     M36  ; 报警
8536  LDF     M612  ; X12-急停
      RST     M11  ; 蜂鸣器
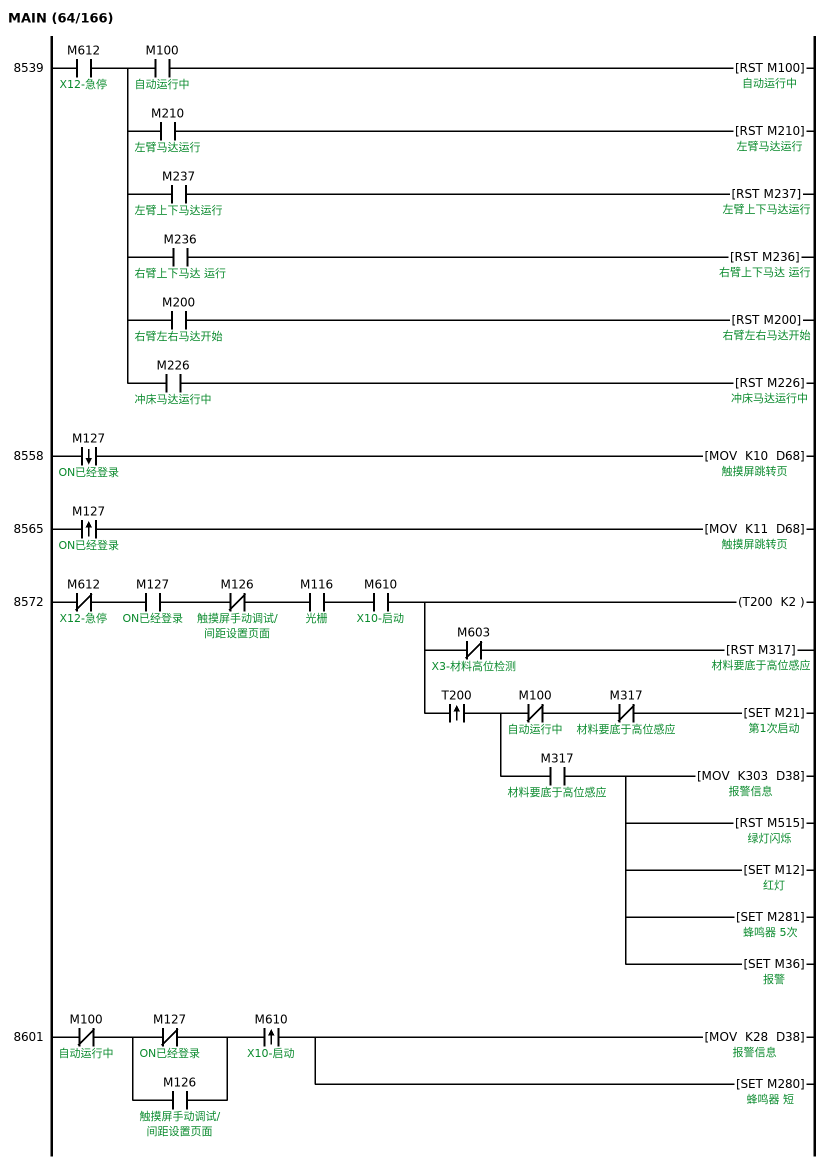
8539  LD      M612  ; X12-急停
      MPS
      AND     M100  ; 自动运行中
      RST     M100  ; 自动运行中
      MRD
      AND     M210  ; 左臂马达运行
      RST     M210  ; 左臂马达运行
      MRD
      AND     M237  ; 左臂上下马达运行
      RST     M237  ; 左臂上下马达运行
      MRD
      AND     M236  ; 右臂上下马达 运行
      RST     M236  ; 右臂上下马达 运行
      MRD
      AND     M200  ; 右臂左右马达开始
      RST     M200  ; 右臂左右马达开始
      MPP
      AND     M226  ; 冲床马达运行中
      RST     M226  ; 冲床马达运行中
8558  LDF     M127  ; ON已经登录
      MOV     K10 D68  ; 触摸屏跳转页
8565  LDP     M127  ; ON已经登录
      MOV     K11 D68
8572  LDI     M612  ; X12-急停
      AND     M127  ; ON已经登录
      ANI     M126  ; 触摸屏手动调试/间距设置页面
      AND     M116  ; 光栅
      AND     M610  ; X10-启动
      OUT     T200 K2
      MPS
      ANI     M603  ; X3-材料高位检测
      RST     M317  ; 材料要底于高位感应
      MPP
      ANDP    T200
      MPS
      ANI     M100  ; 自动运行中
      ANI     M317  ; 材料要底于高位感应
      SET     M21  ; 第1次启动
      MPP
      AND     M317  ; 材料要底于高位感应
      MOV     K303 D38
      RST     M515  ; 绿灯闪烁
      SET     M12  ; 红灯
      SET     M281  ; 蜂鸣器 5次
      SET     M36  ; 报警
8601  LDI     M100  ; 自动运行中
      LDI     M127  ; ON已经登录
      OR      M126  ; 触摸屏手动调试/间距设置页面
      ANB
      ANDP    M610  ; X10-启动
      MOV     K28 D38
      SET     M280  ; 蜂鸣器 短
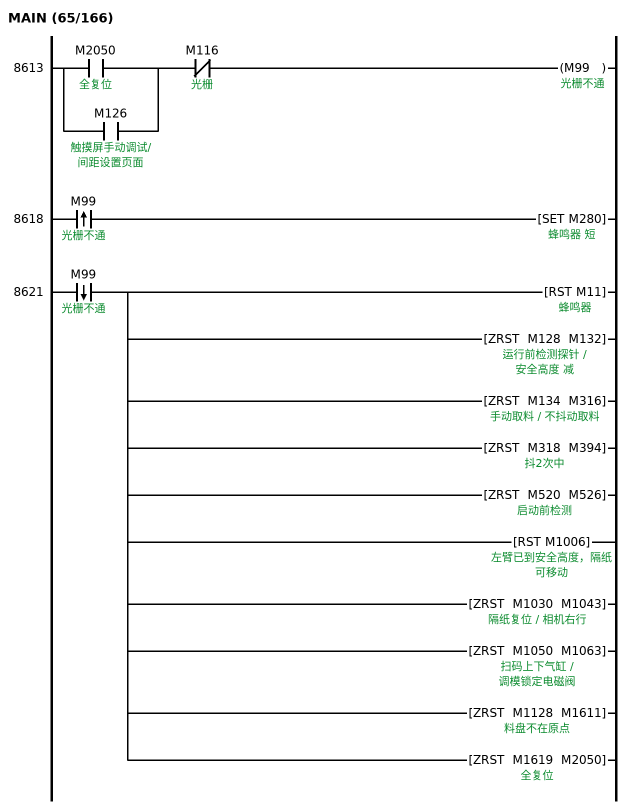
8613  LD      M2050  ; 全复位
      OR      M126  ; 触摸屏手动调试/间距设置页面
      ANI     M116  ; 光栅
      OUT     M99  ; 光栅不通
8618  LDP     M99  ; 光栅不通
      SET     M280  ; 蜂鸣器 短
8621  LDF     M99  ; 光栅不通
      RST     M11  ; 蜂鸣器
      ZRST    M128 M132
      ZRST    M134 M316
      ZRST    M318 M394
      ZRST    M520 M526
      RST     M1006  ; 左臂已到安全高度，隔纸可移动
      ZRST    M1030 M1043
      ZRST    M1050 M1063
      ZRST    M1128 M1611  ; 料盘不在原点
      ZRST    M1619 M2050
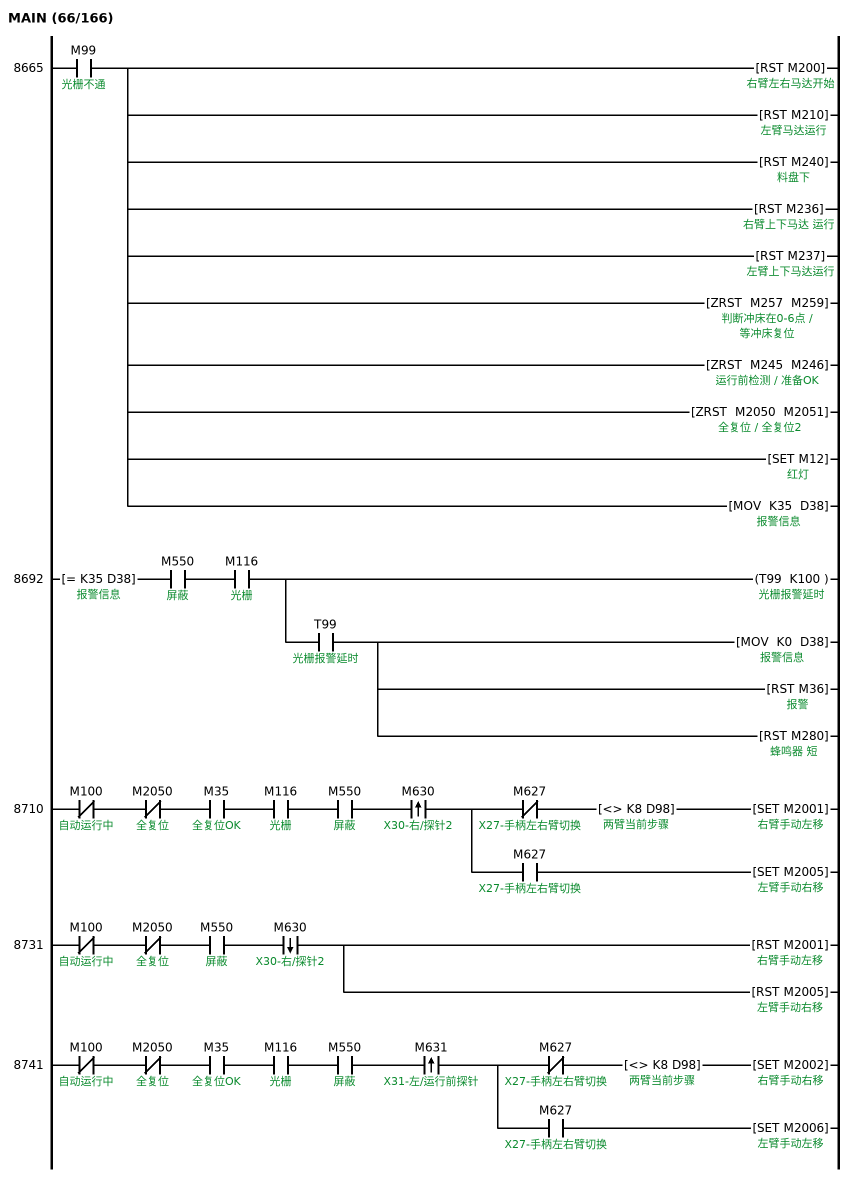
8665  LD      M99  ; 光栅不通
      RST     M200  ; 右臂左右马达开始
      RST     M210  ; 左臂马达运行
      RST     M240  ; 料盘下
      RST     M236  ; 右臂上下马达 运行
      RST     M237  ; 左臂上下马达运行
      ZRST    M257 M259
      ZRST    M245 M246
      ZRST    M2050 M2051
      SET     M12  ; 红灯
      MOV     K35 D38
8692  LD=     K35 D38  ; 报警信息
      AND     M550  ; 屏蔽
      AND     M116  ; 光栅
      OUT     T99 K100  ; 光栅报警延时
      AND     T99  ; 光栅报警延时
      MOV     K0 D38
      RST     M36  ; 报警
      RST     M280  ; 蜂鸣器 短
8710  LDI     M100  ; 自动运行中
      ANI     M2050  ; 全复位
      AND     M35  ; 全复位OK
      AND     M116  ; 光栅
      AND     M550  ; 屏蔽
      ANDP    M630  ; X30-右/探针2
      MPS
      ANI     M627  ; X27-手柄左右臂切换
      AND<>   K8 D98  ; 两臂当前步骤
      SET     M2001  ; 右臂手动左移
      MPP
      AND     M627  ; X27-手柄左右臂切换
      SET     M2005  ; 左臂手动右移
8731  LDI     M100  ; 自动运行中
      ANI     M2050  ; 全复位
      AND     M550  ; 屏蔽
      ANDF    M630  ; X30-右/探针2
      RST     M2001  ; 右臂手动左移
      RST     M2005  ; 左臂手动右移
8741  LDI     M100  ; 自动运行中
      ANI     M2050  ; 全复位
      AND     M35  ; 全复位OK
      AND     M116  ; 光栅
      AND     M550  ; 屏蔽
      ANDP    M631  ; X31-左/运行前探针
      MPS
      ANI     M627  ; X27-手柄左右臂切换
      AND<>   K8 D98  ; 两臂当前步骤
      SET     M2002  ; 右臂手动右移
      MPP
      AND     M627  ; X27-手柄左右臂切换
      SET     M2006  ; 左臂手动左移
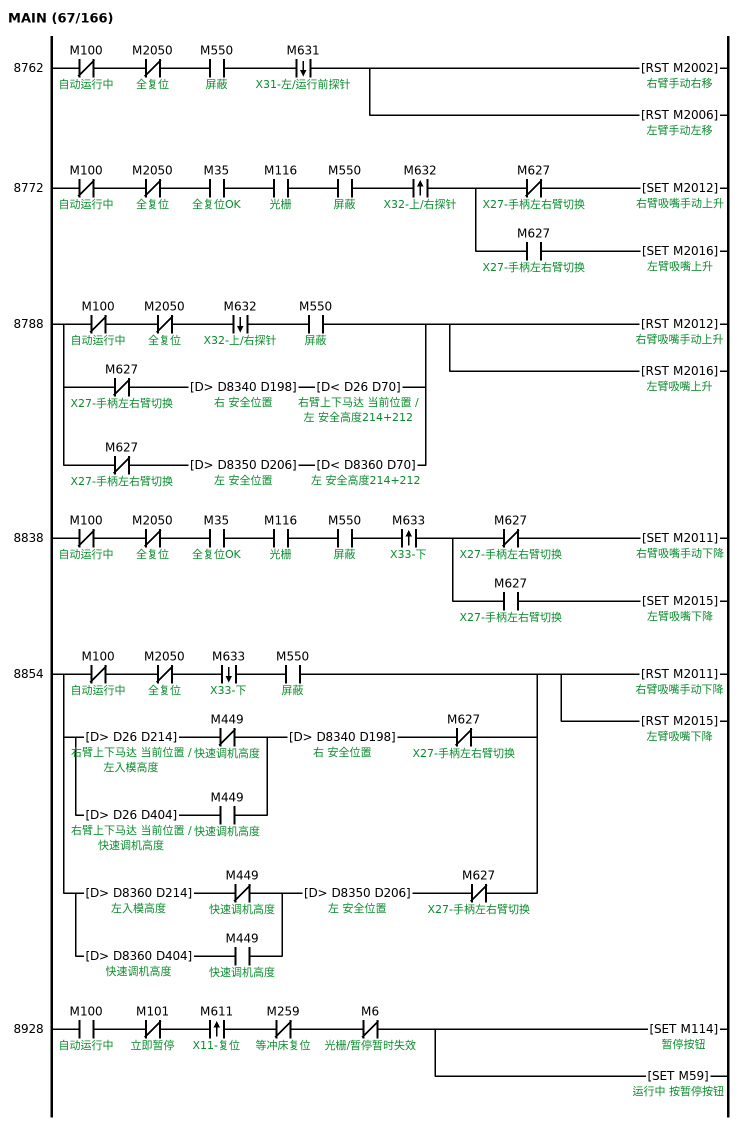
8762  LDI     M100  ; 自动运行中
      ANI     M2050  ; 全复位
      AND     M550  ; 屏蔽
      ANDF    M631  ; X31-左/运行前探针
      RST     M2002  ; 右臂手动右移
      RST     M2006  ; 左臂手动左移
8772  LDI     M100  ; 自动运行中
      ANI     M2050  ; 全复位
      AND     M35  ; 全复位OK
      AND     M116  ; 光栅
      AND     M550  ; 屏蔽
      ANDP    M632  ; X32-上/右探针
      MPS
      ANI     M627  ; X27-手柄左右臂切换
      SET     M2012  ; 右臂吸嘴手动上升
      MPP
      AND     M627  ; X27-手柄左右臂切换
      SET     M2016  ; 左臂吸嘴上升
8788  LDI     M100  ; 自动运行中
      ANI     M2050  ; 全复位
      ANDF    M632  ; X32-上/右探针
      AND     M550  ; 屏蔽
      LDI     M627  ; X27-手柄左右臂切换
      ANDD>   D8340 D198  ; 右 安全位置
      ANDD<   D26 D70  ; 右臂上下马达 当前位置 / 左 安全高度214+212
      ORB
      LDI     M627  ; X27-手柄左右臂切换
      ANDD>   D8350 D206  ; 左 安全位置
      ANDD<   D8360 D70  ; 左 安全高度214+212
      ORB
      RST     M2012  ; 右臂吸嘴手动上升
      RST     M2016  ; 左臂吸嘴上升
8838  LDI     M100  ; 自动运行中
      ANI     M2050  ; 全复位
      AND     M35  ; 全复位OK
      AND     M116  ; 光栅
      AND     M550  ; 屏蔽
      ANDP    M633  ; X33-下
      MPS
      ANI     M627  ; X27-手柄左右臂切换
      SET     M2011  ; 右臂吸嘴手动下降
      MPP
      AND     M627  ; X27-手柄左右臂切换
      SET     M2015  ; 左臂吸嘴下降
8854  LDI     M100  ; 自动运行中
      ANI     M2050  ; 全复位
      ANDF    M633  ; X33-下
      AND     M550  ; 屏蔽
      LDD>    D26 D214  ; 右臂上下马达 当前位置 / 左入模高度
      ANI     M449  ; 快速调机高度
      LDD>    D26 D404  ; 右臂上下马达 当前位置 / 快速调机高度
      AND     M449  ; 快速调机高度
      ORB
      ANDD>   D8340 D198  ; 右 安全位置
      ANI     M627  ; X27-手柄左右臂切换
      ORB
      LDD>    D8360 D214  ; 左入模高度
      ANI     M449  ; 快速调机高度
      LDD>    D8360 D404  ; 快速调机高度
      AND     M449  ; 快速调机高度
      ORB
      ANDD>   D8350 D206  ; 左 安全位置
      ANI     M627  ; X27-手柄左右臂切换
      ORB
      RST     M2011  ; 右臂吸嘴手动下降
      RST     M2015  ; 左臂吸嘴下降
8928  LD      M100  ; 自动运行中
      ANI     M101  ; 立即暂停
      ANDP    M611  ; X11-复位
      ANI     M259  ; 等冲床复位
      ANI     M6  ; 光栅/暂停暂时失效
      SET     M114  ; 暂停按钮
      SET     M59  ; 运行中 按暂停按钮
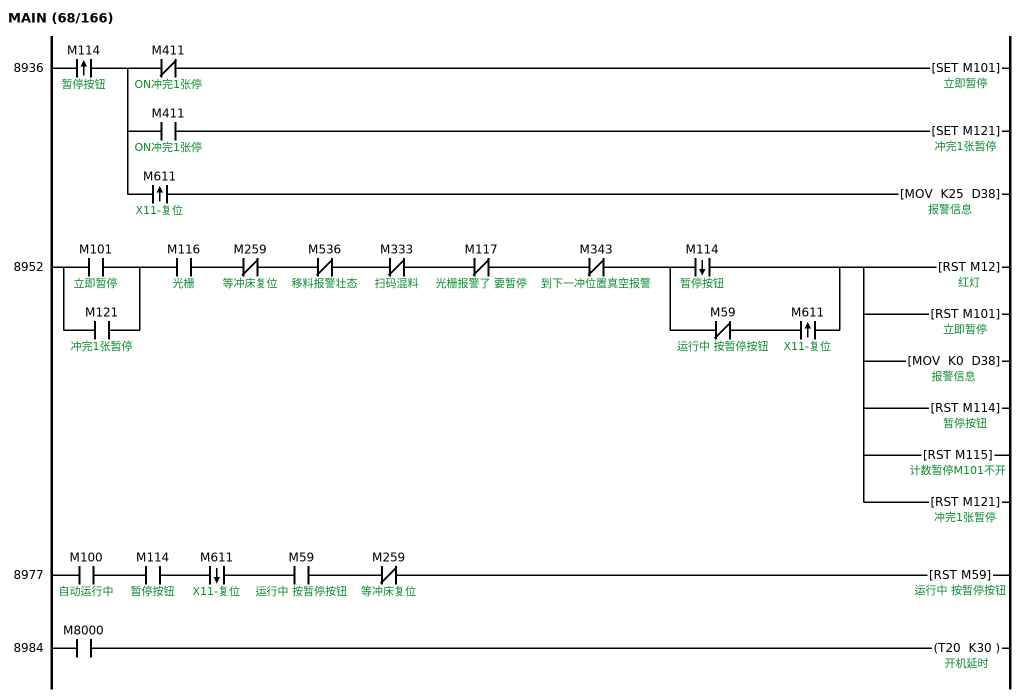
8936  LDP     M114  ; 暂停按钮
      MPS
      ANI     M411  ; ON冲完1张停
      SET     M101  ; 立即暂停
      MRD
      AND     M411  ; ON冲完1张停
      SET     M121  ; 冲完1张暂停
      MPP
      ANDP    M611  ; X11-复位
      MOV     K25 D38
8952  LD      M101  ; 立即暂停
      OR      M121  ; 冲完1张暂停
      AND     M116  ; 光栅
      ANI     M259  ; 等冲床复位
      ANI     M536  ; 移料报警壮态
      ANI     M333  ; 扫码混料
      ANI     M117  ; 光栅报警了 要暂停
      ANI     M343  ; 到下一冲位置真空报警
      LDF     M114  ; 暂停按钮
      LDI     M59  ; 运行中 按暂停按钮
      ANDP    M611  ; X11-复位
      ORB
      ANB
      RST     M12  ; 红灯
      RST     M101  ; 立即暂停
      MOV     K0 D38
      RST     M114  ; 暂停按钮
      RST     M115  ; 计数暂停M101不开
      RST     M121  ; 冲完1张暂停
8977  LD      M100  ; 自动运行中
      AND     M114  ; 暂停按钮
      ANDF    M611  ; X11-复位
      AND     M59  ; 运行中 按暂停按钮
      ANI     M259  ; 等冲床复位
      RST     M59  ; 运行中 按暂停按钮
8984  LD      M8000
      OUT     T20 K30  ; 开机延时
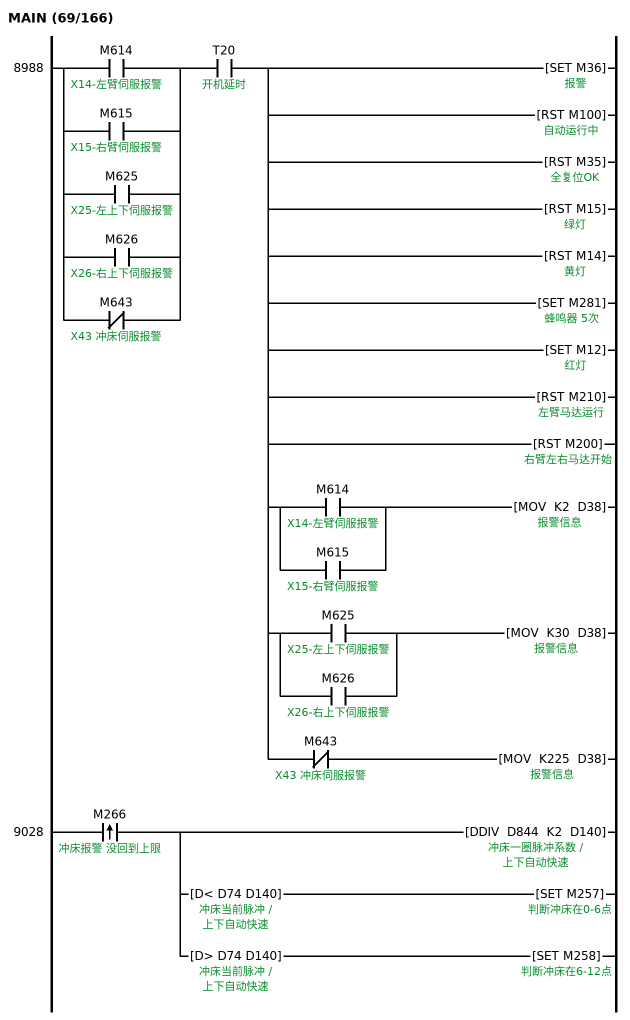
8988  LD      M614  ; X14-左臂伺服报警
      OR      M615  ; X15-右臂伺服报警
      OR      M625  ; X25-左上下伺服报警
      OR      M626  ; X26-右上下伺服报警
      ORI     M643  ; X43 冲床伺服报警
      AND     T20  ; 开机延时
      SET     M36  ; 报警
      RST     M100  ; 自动运行中
      RST     M35  ; 全复位OK
      RST     M15  ; 绿灯
      RST     M14  ; 黄灯
      SET     M281  ; 蜂鸣器 5次
      SET     M12  ; 红灯
      RST     M210  ; 左臂马达运行
      RST     M200  ; 右臂左右马达开始
      MPS
      LD      M614  ; X14-左臂伺服报警
      OR      M615  ; X15-右臂伺服报警
      ANB
      MOV     K2 D38
      MRD
      LD      M625  ; X25-左上下伺服报警
      OR      M626  ; X26-右上下伺服报警
      ANB
      MOV     K30 D38
      MPP
      ANI     M643  ; X43 冲床伺服报警
      MOV     K225 D38
9028  LDP     M266  ; 冲床报警 没回到上限
      DDIV    D844 K2 D140  ; 上下自动快速
      MPS
      ANDD<   D74 D140  ; 冲床当前脉冲 / 上下自动快速
      SET     M257  ; 判断冲床在0-6点
      MPP
      ANDD>   D74 D140  ; 冲床当前脉冲 / 上下自动快速
      SET     M258  ; 判断冲床在6-12点
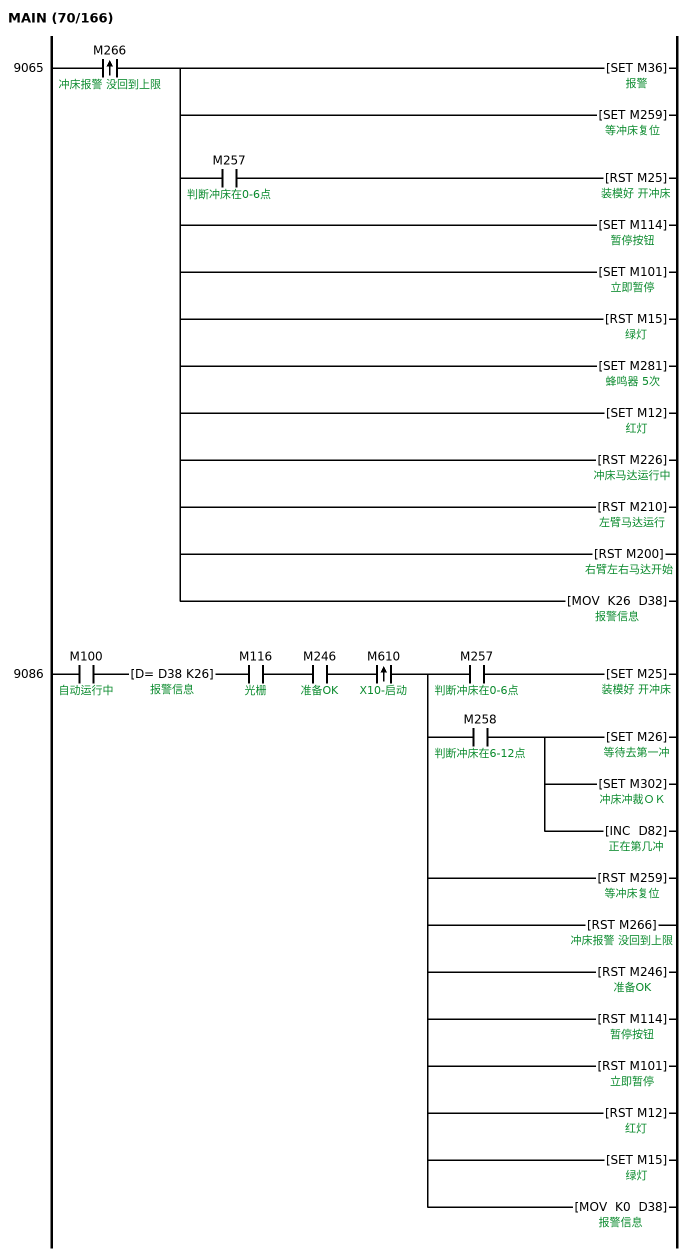
9065  LDP     M266  ; 冲床报警 没回到上限
      SET     M36  ; 报警
      SET     M259  ; 等冲床复位
      MPS
      AND     M257  ; 判断冲床在0-6点
      RST     M25  ; 装模好 开冲床
      MPP
      SET     M114  ; 暂停按钮
      SET     M101  ; 立即暂停
      RST     M15  ; 绿灯
      SET     M281  ; 蜂鸣器 5次
      SET     M12  ; 红灯
      RST     M226  ; 冲床马达运行中
      RST     M210  ; 左臂马达运行
      RST     M200  ; 右臂左右马达开始
      MOV     K26 D38
9086  LD      M100  ; 自动运行中
      ANDD=   D38 K26  ; 报警信息
      AND     M116  ; 光栅
      AND     M246  ; 准备OK
      ANDP    M610  ; X10-启动
      MPS
      AND     M257  ; 判断冲床在0-6点
      SET     M25  ; 装模好 开冲床
      MRD
      AND     M258  ; 判断冲床在6-12点
      SET     M26  ; 等待去第一冲
      SET     M302  ; 冲床冲裁ＯＫ
      INC     D82
      MPP
      RST     M259  ; 等冲床复位
      RST     M266  ; 冲床报警 没回到上限
      RST     M246  ; 准备OK
      RST     M114  ; 暂停按钮
      RST     M101  ; 立即暂停
      RST     M12  ; 红灯
      SET     M15  ; 绿灯
      MOV     K0 D38
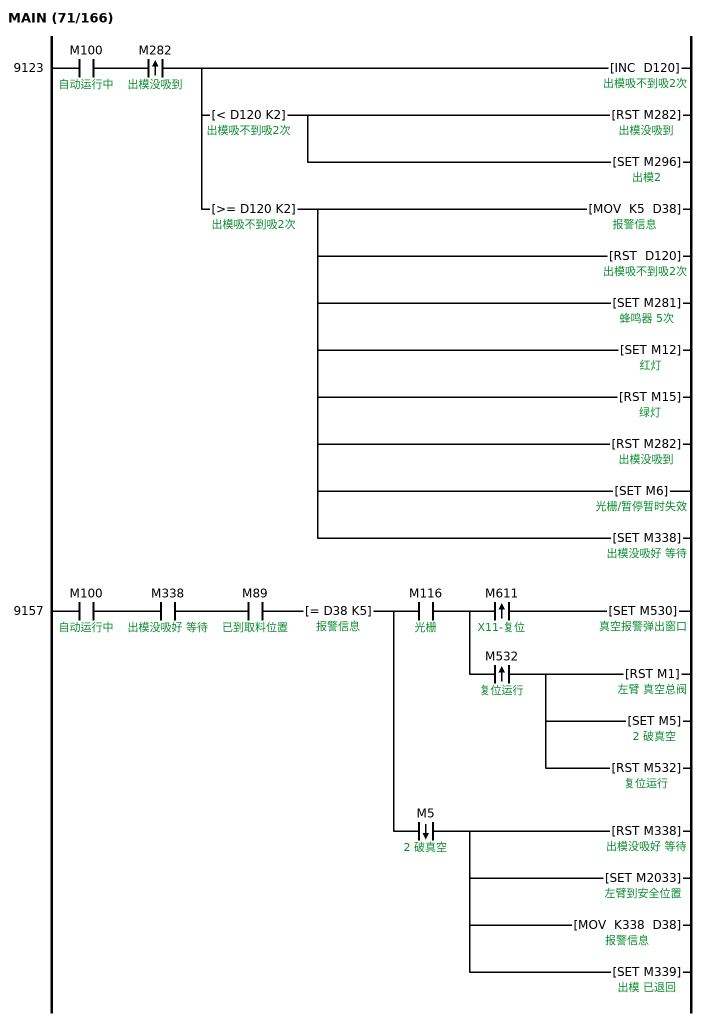
9123  LD      M100  ; 自动运行中
      ANDP    M282  ; 出模没吸到
      INC     D120  ; 出模吸不到吸2次
      MPS
      AND<    D120 K2  ; 出模吸不到吸2次
      RST     M282  ; 出模没吸到
      SET     M296  ; 出模2
      MPP
      AND>=   D120 K2  ; 出模吸不到吸2次
      MOV     K5 D38
      RST     D120  ; 出模吸不到吸2次
      SET     M281  ; 蜂鸣器 5次
      SET     M12  ; 红灯
      RST     M15  ; 绿灯
      RST     M282  ; 出模没吸到
      SET     M6  ; 光栅/暂停暂时失效
      SET     M338  ; 出模没吸好 等待
9157  LD      M100  ; 自动运行中
      AND     M338  ; 出模没吸好 等待
      AND     M89  ; 已到取料位置
      AND=    D38 K5  ; 报警信息
      MPS
      AND     M116  ; 光栅
      MPS
      ANDP    M611  ; X11-复位
      SET     M530  ; 真空报警弹出窗口
      MPP
      ANDP    M532  ; 复位运行
      RST     M1  ; 左臂 真空总阀
      SET     M5  ; 2 破真空
      RST     M532  ; 复位运行
      MPP
      ANDF    M5  ; 2 破真空
      RST     M338  ; 出模没吸好 等待
      SET     M2033  ; 左臂到安全位置
      MOV     K338 D38
      SET     M339  ; 出模 已退回
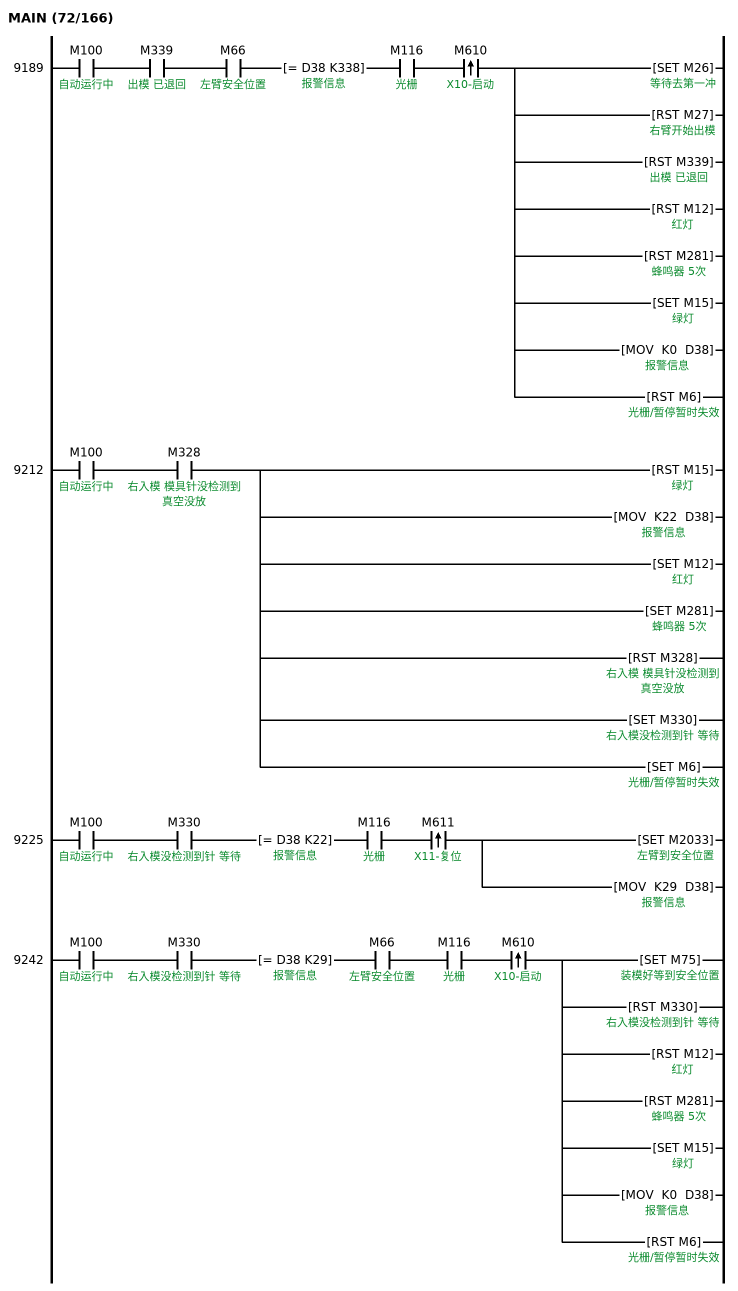
9189  LD      M100  ; 自动运行中
      AND     M339  ; 出模 已退回
      AND     M66  ; 左臂安全位置
      AND=    D38 K338  ; 报警信息
      AND     M116  ; 光栅
      ANDP    M610  ; X10-启动
      SET     M26  ; 等待去第一冲
      RST     M27  ; 右臂开始出模
      RST     M339  ; 出模 已退回
      RST     M12  ; 红灯
      RST     M281  ; 蜂鸣器 5次
      SET     M15  ; 绿灯
      MOV     K0 D38
      RST     M6  ; 光栅/暂停暂时失效
9212  LD      M100  ; 自动运行中
      AND     M328  ; 右入模 模具针没检测到 真空没放
      RST     M15  ; 绿灯
      MOV     K22 D38
      SET     M12  ; 红灯
      SET     M281  ; 蜂鸣器 5次
      RST     M328  ; 右入模 模具针没检测到 真空没放
      SET     M330  ; 右入模没检测到针 等待
      SET     M6  ; 光栅/暂停暂时失效
9225  LD      M100  ; 自动运行中
      AND     M330  ; 右入模没检测到针 等待
      AND=    D38 K22  ; 报警信息
      AND     M116  ; 光栅
      ANDP    M611  ; X11-复位
      SET     M2033  ; 左臂到安全位置
      MOV     K29 D38
9242  LD      M100  ; 自动运行中
      AND     M330  ; 右入模没检测到针 等待
      AND=    D38 K29  ; 报警信息
      AND     M66  ; 左臂安全位置
      AND     M116  ; 光栅
      ANDP    M610  ; X10-启动
      SET     M75  ; 装模好等到安全位置
      RST     M330  ; 右入模没检测到针 等待
      RST     M12  ; 红灯
      RST     M281  ; 蜂鸣器 5次
      SET     M15  ; 绿灯
      MOV     K0 D38
      RST     M6  ; 光栅/暂停暂时失效
